// TIA Portal V17 export
// export: Created 2026-07-16T05:46:42.1531902Z, ExportSetting WithDefaults, DisplayName Totally Integrated Automation Portal, DisplayVersion V17 Update 7, DisplayName TIA Portal Openness, DisplayVersion V17 Update 7, DisplayName TIA Portal Version Control Interface, DisplayVersion V17, DisplayName SINAMICS Startdrive Advanced, DisplayVersion V17 SP2, DisplayName SINAMICS Startdrive G110M, G120, G120C, G120D, G120P, G115D, DisplayVersion V17 SP2, DisplayName SINAMICS Startdrive G130, G150, S120, S150, SINAMICS MV, S210, DisplayVersion V17 SP2, DisplayName STEP 7 Professional, DisplayVersion V17 Update 7, DisplayName STEP 7 Safety, DisplayVersion V17 Update 6, DisplayName WinCC Advanced, DisplayVersion V17 Update 7
VAR_GLOBAL   // PLC tag table "IO_CC_Cav_A"
   O_CC_Coupelle_Up_Cav_A AT %Q600.7 : Bool;
   I_CC_TyrePresent_Pos_2_Cav_A AT %I600.2 : Bool;
   I_CC_TyrePresent_Pos_3_Cav_A AT %I600.3 : Bool;
   I_CC_TyrePresent_Coupelle_Cav_A AT %I600.0 : Bool;
   I_CC_TyrePresent_Exit_Cav_A AT %I600.1 : Bool;
   I_CC_Coupelle_Low_Cav_A AT %I600.4 : Bool;
   I_CC_Coupelle_High_Cav_A AT %I600.5 : Bool;
   I_CC_Motor_Lototo_Cav_A AT %I600.6 : Bool;
   O_CC_Coupelle_Down_Cav_A AT %Q601.7 : Bool;
   I_CC_TyrePresent_Pos_1_Cav_A AT %I601.0 : Bool;
END_VAR
